# EPICS substitutions: HIFIMAGS/HIFIMAGS-IOC-01App/Db/hifimags_magnet.substitutions
file hifimags_magnet.template {
  pattern
    {P, MAG, PSU_IOC}

    {"\$(P)", "X", "\$(X_IOC)"}
    {"\$(P)", "Y", "\$(Y_IOC)"}
    {"\$(P)", "Z", "\$(Z_IOC)"}
    {"\$(P)", "M", "\$(M_IOC)"}
}
